FUNCTION_BLOCK FB_Scale
VAR_INPUT
	rRawData                   	: LREAL;
	rRawDataLowerOffLimit      	: LREAL;
	rRawDataUpperOffLimit      	: LREAL;
	rScaleDataLowerOffLimit    	: LREAL;
	rScaleDataUpperOffLimit    	: LREAL;
	rY_Intercept				: LREAL;
	
END_VAR
VAR_OUTPUT
	rScaleData					: LREAL;
END_VAR
VAR
	m							: LREAL;
END_VAR

IF (rRawDataUpperOffLimit - rRawDataLowerOffLimit <> 0) THEN
	m								:= (rScaleDataUpperOffLimit - rScaleDataLowerOffLimit )/( rRawDataUpperOffLimit - rRawDataLowerOffLimit);

END_IF

rScaleData						:= ( rRawData * m) + rY_Intercept;

END_FUNCTION_BLOCK

(* stored: Version 1.1.0.1, ProductVersion 3.1.4024.12
   POU FB_Scale: Id {1342ee58-0be6-415a-bc13-c7add60c9f0d}, SpecialFunc None *)
